{attribute 'GeneratedUsingTerminal: EPP7041-1002-0016'}
{attribute addProperty BoxType "EPP7041-1002-0016"}
{attribute addProperty Id "AdsAddrAT %I*AMSADDR8Chn0AT %I*USINT1Chn1AT %I*USINT1StateAT %I*UINT2"}
{attribute addProperty CRC "1698221919"}
{attribute addProperty Size "12"}
TYPE InfoData_6538CF5F :
STRUCT
	{attribute addProperty Name "AdsAddr"}
	AdsAddr AT %I* : AMSADDR;
	{attribute addProperty Name "Chn0"}
	Chn0 AT %I* : USINT;
	{attribute addProperty Name "Chn1"}
	Chn1 AT %I* : USINT;
	{attribute addProperty Name "State"}
	State AT %I* : UINT;
END_STRUCT
END_TYPE

(* stored: Version 1.2.0.0, ProductVersion 3.1.4024.9
   DUT InfoData_6538CF5F: Id {a3d170eb-9b81-4908-a6fc-00da6c678f2d} *)
